// TIA Portal V18 export
FUNCTION "Block_FB" : Void   // FC1, FBD
{ S7_Optimized_Access := 'TRUE' }
// stored: SetENOAutomatically false
   VAR_TEMP
      "A" : Bool;
      "B" : Bool;
      Q : Bool;
   END_VAR
BEGIN

REGION Network 1
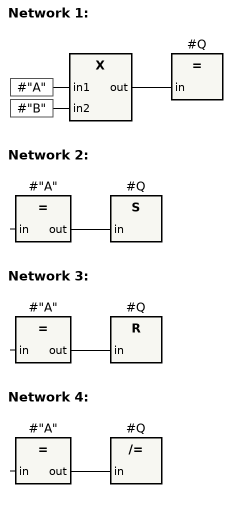
   #Q := #"A" XOR #"B";
END_REGION

REGION Network 2
   #"A" := TRUE;
   #Q := TRUE;
END_REGION

REGION Network 3
   #"A" := TRUE;
   #Q := FALSE;
END_REGION

REGION Network 4
   #"A" := TRUE;
   #Q := NOT TRUE;
END_REGION
END_FUNCTION
